TYPE DUT_RunTime :
STRUCT
	seconds:INT;
	mins:INT;
	hours:DINT;
END_STRUCT
END_TYPE

(* stored: Version 1.1.0.1, ProductVersion 3.1.4024.3
   DUT DUT_RunTime: Id {18a6887a-88b8-4ef0-ac1a-d2568c2dc006} *)
